// TIA Portal V19 export
TYPE "lexchangetray_typeUnEmn_toHandlingXyzFeedback"
// Type: Bool
// stored: Access Published
   STRUCT
      catchEnable : Bool;   // Manual mode parameters for axis control interface
   END_STRUCT;
END_TYPE
